// TIA Portal project "Main" (V16)

(* hardware
DEVICE "S7-1200 station_1"  S7-1200 Station
   slot 0: "Rack_0"  S7-1200 Rack  Rack  V1.0
   slot 1: "PLC_1"  CPU 1212C DC/DC/DC  6ES7 212-1AE40-0XB0  V4.0
*)

// ===== PLC "PLC_1"  CPU 1212C DC/DC/DC =====

VAR_GLOBAL   // PLC tag table "默认变量表"
   "Clock_Byte" AT %MB0 : Byte;
   "Clock_10Hz" AT %M0.0 : Bool;
   "Clock_5Hz" AT %M0.1 : Bool;
   "Clock_2.5Hz" AT %M0.2 : Bool;
   "Clock_2Hz" AT %M0.3 : Bool;
   "Clock_1.25Hz" AT %M0.4 : Bool;
   "Clock_1Hz" AT %M0.5 : Bool;
   "Clock_0.625Hz" AT %M0.6 : Bool;
   "Clock_0.5Hz" AT %M0.7 : Bool;
   "System_Byte" AT %MB1 : Byte;
   "FirstScan" AT %M1.0 : Bool;
   "DiagStatusUpdate" AT %M1.1 : Bool;
   "AlwaysTRUE" AT %M1.2 : Bool;
   "AlwaysFALSE" AT %M1.3 : Bool;
   "Connet" AT %M2.0 : Bool;
   "Run" AT %M2.1 : Bool;
   "Stop" AT %M2.2 : Bool;
   "Q0.0" AT %Q0.0 : Bool;
   "TEST" AT %Q0.1 : Bool;
   "Tag_1" AT %M2.3 : Bool;
END_VAR

DATA_BLOCK "S-Clustr"   // DB4
{ S7_Optimized_Access := 'TRUE' }
VERSION : 0.1
   VAR
      Info : String := '{"TYPE":"PLC-S7-1200"}';
      Info_buff : Array[0..50] of Char;
      Info_Size : UInt;
      Refresh : Array[0..5] of Char;
      recv_buff : Array[0..5] of Char;
      recv : String;
      recv_Size : UInt;
      Device_Status_Run : Int;
      State : Int;
      Stop_command : Char := 'S';
      Run_command_respon : Array[0..2] of Char;
      Stop_command__respon : Array[0..2] of Char;
      led : Byte;
      Run_command : Char := 'R';
      Device_Status_Stop : Int;
   END_VAR
BEGIN
   Stop_command__respon[0] := 'C';
   Stop_command__respon[1] := '$R';
   Stop_command__respon[2] := '$L';
   Run_command_respon[0] := 'O';
   Run_command_respon[1] := '$R';
   Run_command_respon[2] := '$L';
END_DATA_BLOCK

// folder: System blocks/Program resources

DATA_BLOCK "PLC_1_Connection_DB"   // DB2
{ S7_Optimized_Access := 'TRUE' }
AUTHOR : SIMATIC
FAMILY : MC7Plus
NAME : TCON_Prm
VERSION : 1.0
// stored: InstanceOfName TCON_Param
"TCON_Param"
BEGIN
   ID := 1;
   REM_TSAP_ID[1] := B#16#27;
   REM_TSAP_ID[2] := B#16#10;
   REM_STADDR[1] := 192;
   REM_STADDR[2] := 168;
   REM_STADDR[4] := 103;
END_DATA_BLOCK

// folder: (top level)

ORGANIZATION_BLOCK "Main"   // OB1, LAD, ProgramCycle
TITLE = "Main Program Sweep (Cycle)"
{ S7_Optimized_Access := 'TRUE' }
VERSION : 0.1
   VAR_INPUT
      Initial_Call : Bool;   // Initial call of this OB
      Remanence : Bool;   // =True, if remanent data are available
   END_VAR
   VAR_TEMP   // added for the SCL form of the ladder/FBD networks
      _w1 : Bool;
   END_VAR
BEGIN

REGION Network 1
   // 连接服务器
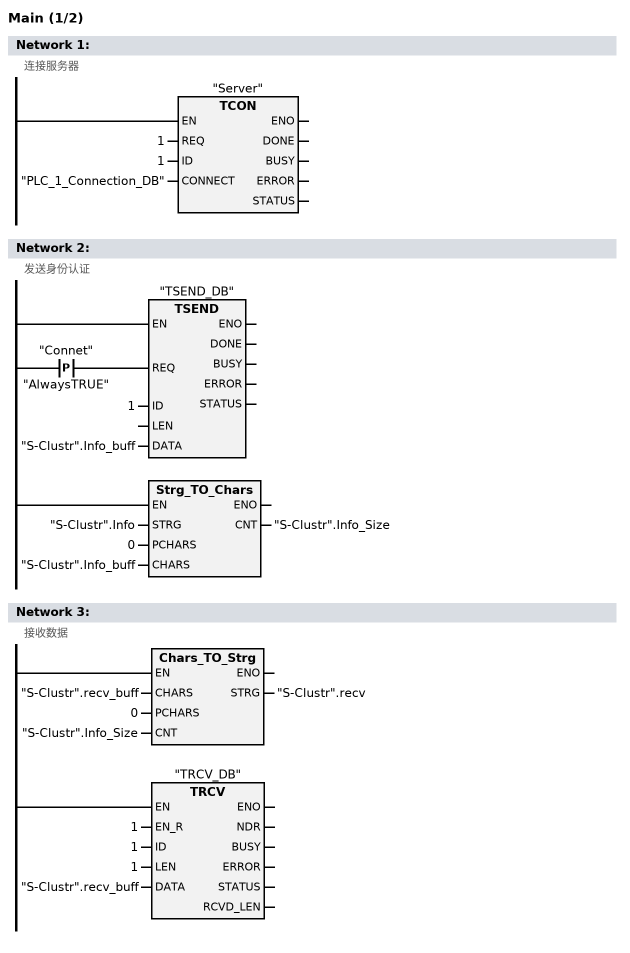
   "Server"(REQ := 1, ID := 1, CONNECT := "PLC_1_Connection_DB");   // TCON
END_REGION

REGION Network 2
   // 发送身份认证
   // no SCL statement known for Strg_TO_Chars: written as a call
   #_w1 := "Connet" AND NOT "AlwaysTRUE";   // rising edge of "Connet"
   "AlwaysTRUE" := "Connet";
   "TSEND_DB"(REQ := #_w1, ID := 1, DATA := "S-Clustr".Info_buff);   // TSEND
   Strg_TO_Chars(Strg := "S-Clustr".Info,
                 pChars := 0,
                 Chars := "S-Clustr".Info_buff,
                 Cnt => "S-Clustr".Info_Size);
END_REGION

REGION Network 3
   // 接收数据
   // no SCL statement known for Chars_TO_Strg: written as a call
   Chars_TO_Strg(Chars := "S-Clustr".recv_buff,
                 pChars := 0,
                 Cnt := "S-Clustr".Info_Size,
                 Strg => "S-Clustr".recv);
   "TRCV_DB"(EN_R := 1, ID := 1, LEN := 1, DATA := "S-Clustr".recv_buff);   // TRCV
END_REGION

REGION Network 4
   // 运行
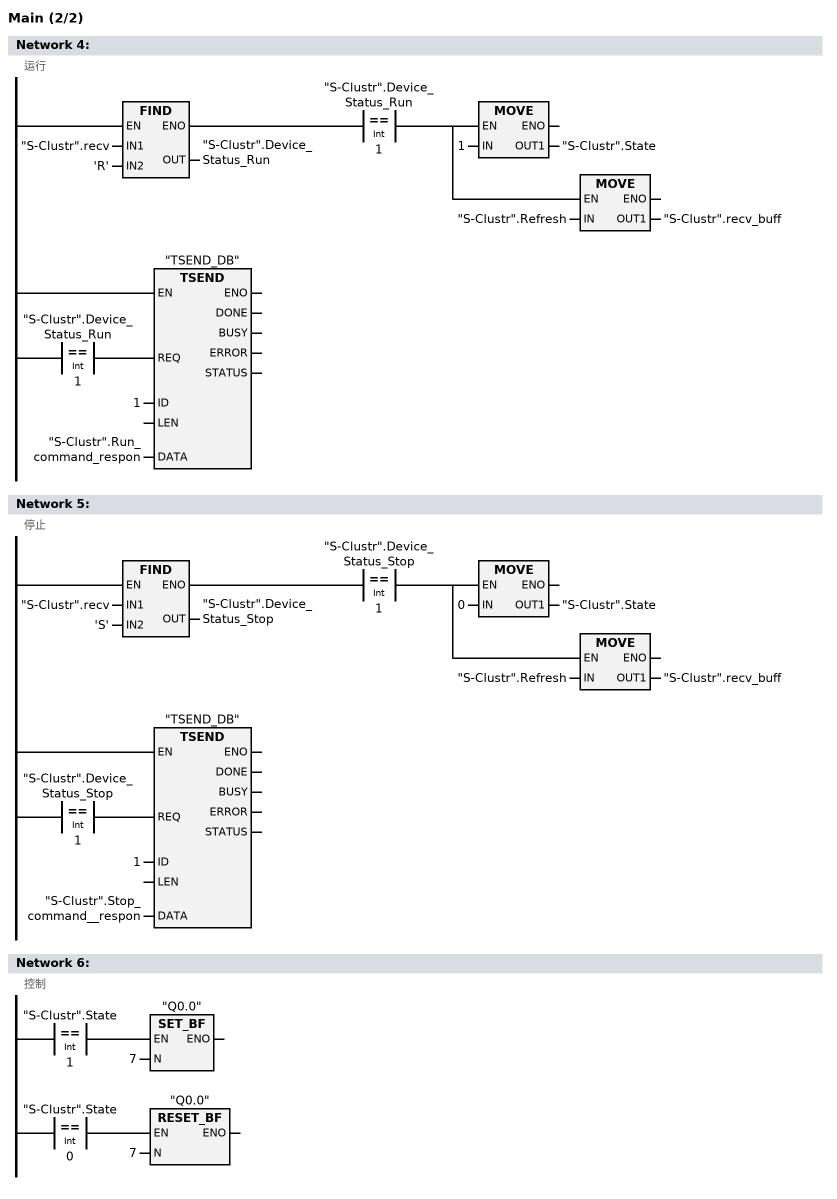
   "S-Clustr".Device_Status_Run := FIND(IN1 := "S-Clustr".recv, IN2 := 'R');
   IF "S-Clustr".Device_Status_Run = 1 THEN
       "S-Clustr".State := 1;
       "S-Clustr".recv_buff := "S-Clustr".Refresh;
   END_IF;
   "TSEND_DB"(REQ := "S-Clustr".Device_Status_Run = 1, ID := 1, DATA := "S-Clustr".Run_command_respon);   // TSEND
END_REGION

REGION Network 5
   // 停止
   "S-Clustr".Device_Status_Stop := FIND(IN1 := "S-Clustr".recv, IN2 := 'S');
   IF "S-Clustr".Device_Status_Stop = 1 THEN
       "S-Clustr".State := 0;
       "S-Clustr".recv_buff := "S-Clustr".Refresh;
   END_IF;
   "TSEND_DB"(REQ := "S-Clustr".Device_Status_Stop = 1, ID := 1, DATA := "S-Clustr".Stop_command__respon);   // TSEND
END_REGION

REGION Network 6
   // 控制
   // no SCL statement known for RBitfield, SBitfield: written as a call
   IF "S-Clustr".State = 1 THEN SET_BF(operand := "Q0.0", n := 7); END_IF;
   IF "S-Clustr".State = 0 THEN RESET_BF(operand := "Q0.0", n := 7); END_IF;
END_REGION
END_ORGANIZATION_BLOCK